TYPE TYP_VALVE_53_HW_OUT :
STRUCT
	CmdHP AT %Q* : BOOL;
	CmdWP AT %Q* : BOOL;
END_STRUCT
END_TYPE

(* stored: Version 1.1.0.1, ProductVersion 3.1.4024.12
   DUT TYP_VALVE_53_HW_OUT: Id {2cc1d54f-5a2c-4467-8ab4-d0ecb27827f0} *)
